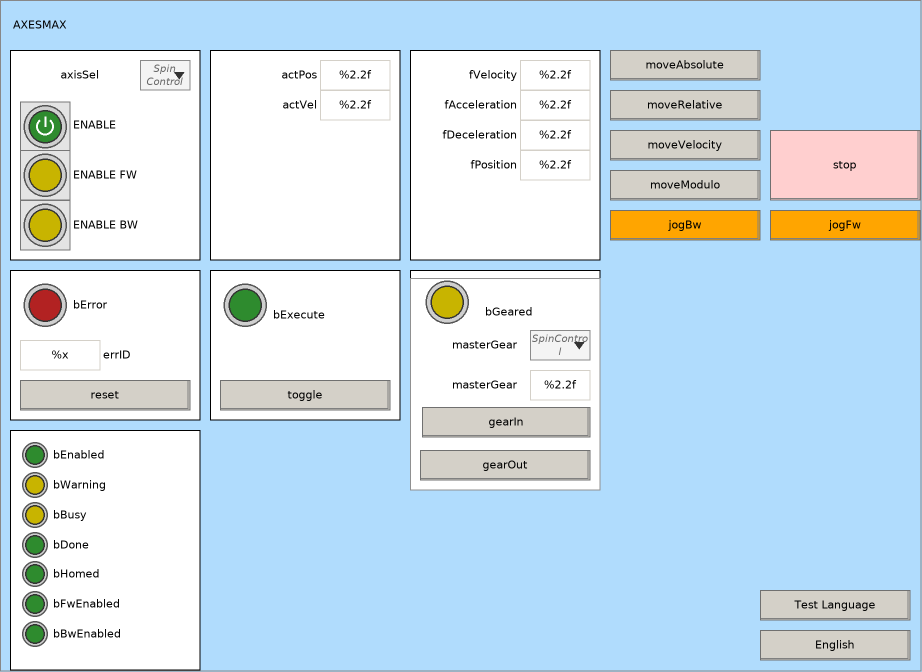
VISUALIZATION MainVisu  // 922x672
    GroupBox (210,270 190x150)
        Rectangle (0,0 190x150)
        Lamp1 (10,10 50x50), variable: GVL.axes[MAIN.hmiAxisSelection].control.bExecute, style: Lamp-Lamp1-Green
        Textfield (60,30 120x30), "bExecute", text list: "languageSupport", text index: "bEexecute"
        Button (10,110 170x30), "toggle", text list: "languageSupport", text index: "toggle"
            OnMouseClick: toggle GVL.axes[MAIN.hmiAxisSelection].control.bExecute
    Rectangle (410,270 190x220)
    GroupBox (10,50 190x210)
        Rectangle (0,0 190x210)
        PowerSwitch (10,50 50x53), variable: GVL.axes[MAIN.hmiAxisSelection].control.bEnable, behaviour: TOGGLE, style: Switch-PowerSwitch-Green
        Textfield (60,50 130x50), "ENABLE", text list: "languageSupport", text index: "enable"
        PushSwitchLed (10,100 50x50), variable: GVL.axes[MAIN.hmiAxisSelection].inputs.bLimitFwd, behaviour: TOGGLE, style: Switch-PushSwitchLed-Yellow
        Textfield (60,100 130x50), "ENABLE FW", text list: "languageSupport", text index: "enFW"
        PushSwitchLed (10,150 50x50), variable: GVL.axes[MAIN.hmiAxisSelection].inputs.bLimitBwd, behaviour: TOGGLE, style: Switch-PushSwitchLed-Yellow
        Textfield (60,150 130x50), "ENABLE BW", text list: "languageSupport", text index: "enBW"
        SpinControl (130,10 50x30), variable: MAIN.hmiAxisSelection
            p651134158: GVL_APP.axisNum
        Textfield (10,10 120x30), "axisSel", text variable: GVL_APP.axisNum, text list: "languageSupport", text index: "axisSel"
    Button (760,590 150x30), "Test Language"
        OnMouseClick: ChangeLanguage ChangeLanguage=Test
    Button (760,630 150x30), "English"
        OnMouseClick: ChangeLanguage ChangeLanguage=default
    Textfield (10,10 190x30), "AXESMAX", text variable: GVL_APP.axisNum, text list: "languageSupport", text index: "axesAvailable"
    Button (610,50 150x30), "moveAbsolute", input disabled if: GVL.axes[MAIN.hmiAxisSelection].status.bGeared, text list: "languageSupport", text index: "moveAbsolute"
        OnMouseClick: execute { GVL.axes[Main.hmiAxisSelection].control.eCommand:=MotionFunctions.MoveAbsolute; GVL.axes[Main.hmiAxisSelection].control.bExecute:=TRUE; }
    Button (610,130 150x30), "moveVelocity", input disabled if: GVL.axes[MAIN.hmiAxisSelection].status.bGeared, text list: "languageSupport", text index: "moveVelocity"
        OnMouseClick: execute { GVL.axes[Main.hmiAxisSelection].control.eCommand:=MotionFunctions.MoveVelocity; GVL.axes[Main.hmiAxisSelection].control.bExecute:=TRUE; }
    Button (610,90 150x30), "moveRelative", input disabled if: GVL.axes[MAIN.hmiAxisSelection].status.bGeared, text list: "languageSupport", text index: "moveRelative"
        OnMouseClick: execute { GVL.axes[Main.hmiAxisSelection].control.eCommand:=MotionFunctions.MoveRelative; GVL.axes[Main.hmiAxisSelection].control.bExecute:=TRUE; }
    Button (610,170 150x30), "moveModulo", input disabled if: GVL.axes[MAIN.hmiAxisSelection].status.bGeared, text list: "languageSupport", text index: "moveModulo"
        OnMouseClick: execute { GVL.axes[Main.hmiAxisSelection].control.eCommand:=MotionFunctions.MoveModulo; GVL.axes[Main.hmiAxisSelection].control.bExecute:=TRUE; }
    Button (770,130 150x70), "stop", pressed state: GVL.axes[Main.hmiAxisSelection].control.bStop, input disabled if: GVL.axes[MAIN.hmiAxisSelection].status.bGeared, text list: "languageSupport", text index: "stop"
        toggle GVL.axes[Main.hmiAxisSelection].control.bStop
    Button (610,210 150x30), "jogBw", input disabled if: GVL.axes[MAIN.hmiAxisSelection].status.bGeared, text list: "languageSupport", text index: "jogBw"
        OnMouseUp: execute { GVL.axes[Main.hmiAxisSelection].control.bJogBwd:= FALSE; }
        OnMouseClick: execute { GVL.axes[Main.hmiAxisSelection].control.eCommand:=MotionFunctions.Jog; }
        OnMouseDown: execute { GVL.axes[Main.hmiAxisSelection].control.bJogBwd:= TRUE; }
    Button (770,210 150x30), "jogFw", input disabled if: GVL.axes[MAIN.hmiAxisSelection].status.bGeared, text list: "languageSupport", text index: "jogFw"
        OnMouseUp: execute { GVL.axes[Main.hmiAxisSelection].control.bJogFwd:= FALSE; }
        OnMouseClick: execute { GVL.axes[Main.hmiAxisSelection].control.eCommand:=MotionFunctions.Jog; }
        OnMouseDown: execute { GVL.axes[Main.hmiAxisSelection].control.bJogFwd:= TRUE; }
    GroupBox (10,270 190x150)
        Rectangle (0,0 190x150)
        Textfield (90,70 90x30), "errID", text list: "languageSupport", text index: "errID"
        Textfield (10,70 80x30), "%x", text variable: GVL.axes[MAIN.hmiAxisSelection].status.nErrorID
        Lamp1 (10,10 50x50), variable: GVL.axes[MAIN.hmiAxisSelection].status.bError, style: Lamp-Lamp1-Red
        Textfield (60,20 120x30), "bError", text list: "languageSupport", text index: "bError"
        Button (10,110 170x30), "reset", pressed state: GVL.axes[Main.hmiAxisSelection].control.bReset, text list: "languageSupport", text index: "reset"
            OnMouseClick: toggle GVL.axes[Main.hmiAxisSelection].control.bReset
    GroupBox (10,430 190x240)
        Rectangle (0,0 190x240)
        Lamp1 (10,10 30x30), variable: GVL.axes[MAIN.hmiAxisSelection].status.bEnabled, style: Lamp-Lamp1-Green
        Textfield (40,10 140x30), "bEnabled", text list: "languageSupport", text index: "bEnabled"
        Lamp1 (10,40 30x30), variable: GVL.axes[MAIN.hmiAxisSelection].status.bWarning, style: Lamp-Lamp1-Yellow
        Textfield (40,40 140x30), "bWarning", text list: "languageSupport", text index: "bWarning"
        Lamp1 (10,70 30x30), variable: GVL.axes[MAIN.hmiAxisSelection].status.bBusy, style: Lamp-Lamp1-Yellow
        Textfield (40,70 140x30), "bBusy", text list: "languageSupport", text index: "bBusy"
        Lamp1 (10,100 30x30), variable: GVL.axes[MAIN.hmiAxisSelection].status.bDone, style: Lamp-Lamp1-Green
        Textfield (40,100 140x30), "bDone", text list: 'languageSupport', text index: "bDone"
        Lamp1 (10,129 30x30), variable: GVL.axes[MAIN.hmiAxisSelection].status.bHomed, style: Lamp-Lamp1-Green
        Textfield (40,129 140x30), "bHomed", text list: "languageSupport", text index: "bHomed"
        Lamp1 (10,159 30x30), variable: GVL.axes[MAIN.hmiAxisSelection].status.bFwEnabled, style: Lamp-Lamp1-Green
        Lamp1 (10,189 30x30), variable: GVL.axes[MAIN.hmiAxisSelection].status.bBwEnabled, style: Lamp-Lamp1-Green
        Textfield (40,159 140x30), "bFwEnabled", text list: "languageSupport", text index: "bFwEnabled"
        Textfield (40,189 140x30), "bBwEnabled", text list: "languageSupport", text index: "bBwEnabled"
    GroupBox (210,50 190x210)
        Rectangle (0,0 190x210)
        Textfield (110,10 70x30), "%2.2f", text variable: GVL.axes[MAIN.hmiAxisSelection].status.fActPosition
        Textfield (10,10 100x30), "actPos", text list: "languageSupport", text index: "actposition"
        Textfield (10,40 100x30), "actVel", text list: "languageSupport", text index: "actVelocity"
        Textfield (110,40 70x30), "%2.2f", text variable: GVL.axes[MAIN.hmiAxisSelection].status.fActVelocity
    GroupBox (410,50 190x210)
        Rectangle (0,0 190x210)
        Textfield (10,10 100x30), "fVelocity", text list: "languageSupport", text index: "fVelocity"
        Textfield (110,10 70x30), "%2.2f", text variable: GVL.axes[MAIN.hmiAxisSelection].config.fVelocity
            OnMouseClick: write GVL.axes[MAIN.hmiAxisSelection].config.fVelocity via Default
        Textfield (10,40 100x30), "fAcceleration", text list: "languageSupport", text index: "fAcceleration"
        Textfield (110,40 70x30), "%2.2f", text variable: GVL.axes[MAIN.hmiAxisSelection].config.fAcceleration
            OnMouseClick: write GVL.axes[MAIN.hmiAxisSelection].config.fAcceleration via Default
        Textfield (10,70 100x30), "fDeceleration", text list: "languageSupport", text index: "fDeceleration"
        Textfield (110,70 70x30), "%2.2f", text variable: GVL.axes[MAIN.hmiAxisSelection].config.fDeceleration
            OnMouseClick: write GVL.axes[MAIN.hmiAxisSelection].config.fDeceleration via Default
        Textfield (10,100 100x30), "fPosition", text list: "languageSupport", text index: "fPosition"
        Textfield (110,100 70x30), "%2.2f", text variable: GVL.axes[MAIN.hmiAxisSelection].config.fPosition
            OnMouseClick: write GVL.axes[MAIN.hmiAxisSelection].config.fPosition via Default
    GroupBox (410,270 190x220)
        Lamp1 (12,7 50x50), variable: GVL.axes[MAIN.hmiAxisSelection].status.bGeared, style: Lamp-Lamp1-Yellow
        Textfield (72,27 120x30), "bGeared", text list: "languageSupport", text index: "bGeared"
        SpinControl (120,60 60x30), variable: GVL.axes[MAIN.hmiAxisSelection].masterAxis.index
            p651134158: GVL_APP.axisNum
        Textfield (10,60 100x30), "masterGear", text list: "languageSupport", text index: "masterGear"
        Textfield (120,100 60x30), "%2.2f", text variable: GVL.axes[MAIN.hmiAxisSelection].masterAxis.ratio
            OnMouseClick: write GVL.axes[MAIN.hmiAxisSelection].masterAxis.ratio via Default
        Textfield (10,100 100x30), "masterGear", text list: "languageSupport", text index: "gearRatio"
        Button (12,137 168x30), "gearIn", text list: "languageSupport", text index: "gearIn"
            OnMouseClick: execute { GVL.axes[Main.hmiAxisSelection].control.eCommand:=MotionFunctions.GearIn; GVL.axes[Main.hmiAxisSelection].control.bExecute:=TRUE; }
        Button (10,180 170x30), "gearOut", text list: "languageSupport", text index: "gearOut"
            OnMouseClick: execute { GVL.axes[Main.hmiAxisSelection].control.eCommand:=MotionFunctions.GearOut; GVL.axes[Main.hmiAxisSelection].control.bExecute:=TRUE; }
END_VISUALIZATION

(* stored: Version 1.1.0.1, ProductVersion 3.1.4024.0
   Visu MainVisu: Id {98c8ae72-e756-4d11-b6a5-5914882e2424} *)
